FUNCTION_BLOCK ABSTRACT FB_UniversalModbusSlave IMPLEMENTS I_UniversalModbusSlave
VAR
	bFirstCycle : BOOL := TRUE;
	sName : STRING;
	iUnitID : BYTE;
	bError : BOOL; //Device Error
	bModbusError : BOOL;// Modbus Communication error
	bReallyError : BOOL;
	tonConfirmReallyError : TON;
	timeConfirmReallyError : TIME := T#15S;
	arrAddressRead : ARRAY [0..50] OF ARRAY [0..2] OF WORD;
	(*arrAddressRead[x][y]: +x : index of Region Read.  arrAddressRead[0]: the first region Read.
							+y:
								case y of
									0: Register address for Read
									1: Number of register for read
									2: Function Read
					 *)
	iNumAddRegionRead : UINT;
	
	arrAddressWrite	 : ARRAY [0..20] OF ARRAY [0..10] OF WORD;// write Multiple or single register
	(* the 20 is max number of region write,
		arrAddressWrite[x][y] : +x: index of Region Read.  arrAddressRead[0]: the first region Read. 
								+y:
									case y of
										0 :  Register address for Write
										1 : number of register will be write => modbus master automatic choose Function Write( single Register or Multi Regiseter)
										2..9 : max 8 value for write
										10: Write Function : e.g E_ModbusFunction.WriteSingleCoil
															
	*)
	iNumAddRegionWrite	: UINT;

	
END_VAR

PROPERTY AddressRead : POINTER TO WORD
GET
AddressRead := ADR(arrAddressRead);
END_GET
END_PROPERTY

PROPERTY AddressWrite : POINTER TO WORD
GET
AddressWrite := ADR( arrAddressWrite);
END_GET
END_PROPERTY

METHOD Convert : BOOL
VAR_INPUT
	iRegionNo	:	INT;
	pReadData	:	POINTER TO word;
END_VAR
END_METHOD

PROPERTY Error : Reference to Bool
GET
Error ref= bError;
END_GET
END_PROPERTY

METHOD FirstCycle
VAR_INPUT
	sName : STRING;
	iUnitID : BYTE ; 		//modbus address of the device : 1- 255
END_VAR
THIS^.sName := sName;
THIS^.iUnitID := iUnitID;
END_METHOD

PROPERTY ModbusError : Reference to bool
GET
ModbusError REF= bModbusError;
END_GET
END_PROPERTY

PROPERTY Name : STRING
GET
Name := sName;
END_GET
SET
sName := Name;
END_SET
END_PROPERTY

PROPERTY NumAddRegionRead : UINT
GET
NumAddRegionRead := iNumAddRegionRead;
END_GET
END_PROPERTY

PROPERTY NumAddRegionWrite : UINT
GET
NumAddRegionWrite := iNumAddRegionWrite;
END_GET
END_PROPERTY

(*if Error(from device) or ModbusError(from Modbus Communicate) Remain in TimeRemainConfirmReallyError)
 |ReallyError is TRUE
 |Implement depending on derived FB (Extended FB)
 |Example of Implement:
 		tonConfirmReallyError(
			IN := bError OR iModbusErrorID <> MODBUS_ERRORS,
			PT := timeConfirmReallyError,
			Q => bReallyError 
		);
*)
PROPERTY ReallyError : REFERENCE to bool
GET
ReallyError ref= bReallyError;
END_GET
END_PROPERTY

PROPERTY TimeRemainConfirmReallyError : Time
GET
TimeRemainConfirmReallyError := timeConfirmReallyError;
END_GET
SET
timeConfirmReallyError := TimeRemainConfirmReallyError;
END_SET
END_PROPERTY

(*
|ID address : 0-255
*)
PROPERTY UnitID : BYTE
GET
UnitID := iUnitID;
END_GET
SET
iUnitID := UnitID;
END_SET
END_PROPERTY

END_FUNCTION_BLOCK

(* stored: Version 1.1.0.1, ProductVersion 3.1.4024.12
   POU FB_UniversalModbusSlave: Id {e818357c-5cba-48ce-9997-4578111a52fe}, SpecialFunc None
   Property AddressRead: Id {6bad1251-2173-4dad-ba55-b0ca54c51b4b}
   Get Get: Id {985bce2e-167a-45be-8089-4bec8ed22891}
   Property AddressWrite: Id {5c4258fd-a88b-4ea9-9dad-ce3ab400d74c}
   Get Get: Id {a0e8c4bf-b72b-4849-87ca-51e8c4ef32ff}
   Method Convert: Id {3fd4f7ca-261b-4d44-a547-551bb3314b31}
   Property Error: Id {da66706d-9d45-4a14-ba51-81c50c8658c2}
   Get Get: Id {bb7c85a9-0bd8-4d99-9cd5-0d041702dbea}
   Method FirstCycle: Id {5bee89eb-ef51-45da-b0f8-e42cc2ee867a}
   Property ModbusError: Id {35fd54f6-a793-47c3-b175-f93b571c04d9}
   Get Get: Id {7135c6e3-59dc-4401-9c16-e08930a23d1d}
   Property Name: Id {06664f22-c56c-4b15-a1d7-a34951a97f8f}
   Get Get: Id {9022ba2a-8142-4b11-aa2b-314496623ffe}
   Set Set: Id {6f38bf1f-ebc9-4220-aa3d-695fb0fa3d27}
   Property NumAddRegionRead: Id {b5abfa30-10e8-4954-8477-81f742d0936e}
   Get Get: Id {f25e2842-516b-4ae1-85e4-95db72ca8802}
   Property NumAddRegionWrite: Id {969a2335-93c3-4c90-91d6-c32d995f4ac2}
   Get Get: Id {b1adea90-2fa2-4e92-a2fc-89d69ec231dc}
   Property ReallyError: Id {55cab104-0dd6-49f6-b898-9d9a68d90f06}
   Get Get: Id {7e199315-13d6-4777-9c2b-a59390e99f40}
   Property TimeRemainConfirmReallyError: Id {4b485358-80eb-41c1-9512-5ba8fd99477f}
   Get Get: Id {af2f17a0-7873-4ac1-8c9b-f63e9b80aca0}
   Set Set: Id {426bd8e0-651c-4d97-82cd-9ee9c4e0cf6e}
   Property UnitID: Id {09876766-f5af-4b25-9fd2-4a972765efd0}
   Get Get: Id {cd055b1c-cf68-47e9-b9fd-fac9e0785529}
   Set Set: Id {0fe61a22-da1d-49e5-a05a-46b09e346e4b} *)
